(*======================================================================================================================================*)
(*//=============================================================================\\
||  _   _ _  __  _         _                        _   _                      ||
|| | \ | | |/ / / \  _   _| |_ ___  _ __ ___   __ _| |_(_) ___  _ __         ||
|| |  \| | ' / / _ \| | | | __/ _ \| '_ ` _ \ / _` | __| |/ _ \| '_ \        ||
|| | |\  | . \/ ___ \ |_| | || (_) | | | | | | (_| | |_| | (_) | | | |       ||
|| |_| \_|_|\_\_/  \_\__,_|\__\___/|_| |_| |_|\__,_|\__|_|\___/|_| |_|       ||
||                                                                             ||
\\=============================================================================//
fb_RS485Search:	Suchfunktion um Automatisch alle ID's im Bus zu Scannen*)
(*
Date          	| Version    	| created under        	| Author          	| Remark *)
(*====================================================================================================================================================*)
(*03/06/2025   	| 1.00      		| TC3		  		| N.Kersting       | first release *)
(*====================================================================================================================================================*)
FUNCTION_BLOCK fb_RS485IdScan
VAR_INPUT
	I_bStartSearch		:BOOL;
	I_diStartID			:DINT	:= 5000;
	I_diMaxID			:DINT	:= 6000;
	I_sStartZeichen		:BYTE := 16#FD;										(* Startzeichen Präfix *)
	I_sEndZeichen		:BYTE := 16#FE;										(* Endzeichen Suffix *)
	I_tWait				:TIME := T#300MS;
	I_StringReceived	:STRING(255);
END_VAR
VAR_OUTPUT
	Q_bSend				:BOOL;
	Q_sSearchString		:STRING(255);
	Q_iCnt				:INT;
	Q_sState			:STRING;
	Q_sIDList			:ARRAY[1..cMaxScanIDs] OF DINT;
END_VAR
VAR
	i					:INT;
	iArrIdx				:INT := 1;
	fbPingEvent			:fb_BusPingEvent;
	diActId				:DINT;
	iStep				:INT;
	tonWait				:ton;
	rTrigSearch			:r_trig;
END_VAR


tonWait(
	PT := I_tWait);
	
rTrigSearch(CLK:= I_bStartSearch, Q=> );

IF NOT I_bStartSearch
THEN
	iStep := 0;
END_IF
	
CASE iStep OF
(*=========================================================================*)
0:	Q_sState := 'INIT';
	tonWait.IN := FALSE;
	Q_bSend := FALSE;
	diActId := I_diStartID;
	Q_sSearchString := '';
	iArrIdx := 1;
	Q_iCnt := 0;
	
	IF rTrigSearch.Q
		AND I_diStartID >0
		AND I_diMaxID >0
	THEN
		FOR i := 1 TO cMaxScanIDs BY 1 DO 
			Q_sIDList[i] := 0;
		END_FOR
		
		iStep := iStep +1;
	END_IF
	
(*=========================================================================*)
1:	Q_bSend := FALSE;
	tonWait.IN := FALSE;
	
	IF diActId <= I_diMaxID
	THEN		
		iStep := iStep +1;
	ELSE
		iStep := 0;
	END_IF
	
(*=========================================================================*)
2:	Q_sSearchString := CONCAT(F_ToCHR(I_sStartZeichen),DINT_TO_STRING(diActId));
	Q_sSearchString := CONCAT(Q_sSearchString,'.TMP.1.gSTATUS');
	Q_sSearchString := CONCAT(Q_sSearchString,F_ToCHR(I_sEndZeichen));
	Q_sSearchString := CONCAT(Q_sSearchString,F_ToCHR(I_sStartZeichen));
	Q_sSearchString := CONCAT(Q_sSearchString,DINT_TO_STRING(diActId));
	Q_sSearchString := CONCAT(Q_sSearchString,'.OUT.210.gSTATUS');
	Q_sSearchString := CONCAT(Q_sSearchString,F_ToCHR(I_sEndZeichen));
	
	iStep := iStep +1;
	
(*=========================================================================*)
3:	Q_sState := 'Suchen Aktiv';
	tonWait.IN := TRUE;
	Q_bSend := TRUE;
	
	fbPingEvent(
		I_diID:= 				diActId, 
		I_sReceivedString:= 	I_StringReceived, 
		I_bReset:= ,
		Q_bOut=> );
		
	IF fbPingEvent.Q_bOut
	THEN
		Q_bSend := FALSE;
		iStep := iStep +1;
	ELSIF
		tonWait.Q
	THEN
		Q_bSend := FALSE;
		IF diActId <I_diMaxID
		THEN
			diActId := diActId +1;
			iStep := 1; (* nächsten Teilnehmer Suchen *)
		ELSE
			iStep := 6;	(* Scan Fertig *)
		END_IF
	END_IF
	
(*=========================================================================*)
4:	(* Teilnehmer gefunden ! *)
	Q_sState := 'Teilnehmer gefunden!';
	tonWait.IN := FALSE;	
	Q_bSend := FALSE;
	Q_sIDList[iArrIdx] := diActId;
	
	IF diActId <I_diMaxID
	THEN
		IF iArrIdx < cMaxScanIDs 
		THEN
			diActId := diActId +1;
			iArrIdx := iArrIdx +1;
			iStep := 1; (* nächsten Teilnehmer Suchen *)
		ELSE
			iStep := 5;
		END_IF
	ELSE
		iStep := 6;	(* Scan Fertig *)
	END_IF
	
(*=========================================================================*)
5:	(* Liste Voll! *)
	Q_sState := 'Liste Voll!';
	
(*=========================================================================*)
6:	(* Scan Fertig *)
	Q_iCnt := 0;
	
	FOR i := 1 TO cMaxScanIDs BY 1 DO 
		IF Q_sIDList[i] <> 0
		THEN
			Q_iCnt := Q_iCnt+1;
		END_IF
	END_FOR
	
	Q_sState := CONCAT('Scan Fertig! Es wurden: ',INT_TO_STRING(Q_iCnt));
	Q_sState := CONCAT(Q_sState,' Teilnehmer gefunden!');
		
	IF rTrigSearch.Q
	THEN
		iStep := 0;
	END_IF
END_CASE

END_FUNCTION_BLOCK

(* stored: Version 1.1.0.1, ProductVersion 3.1.4024.16
   POU fb_RS485IdScan: Id {626e2986-02cd-4da6-89a8-c21a082cde8a}, SpecialFunc None *)
